SYSTEM distributed_example
  (* Version 1.0, 2025-11-18, obotnar *)
  APPLICATION distributed_exampleApp
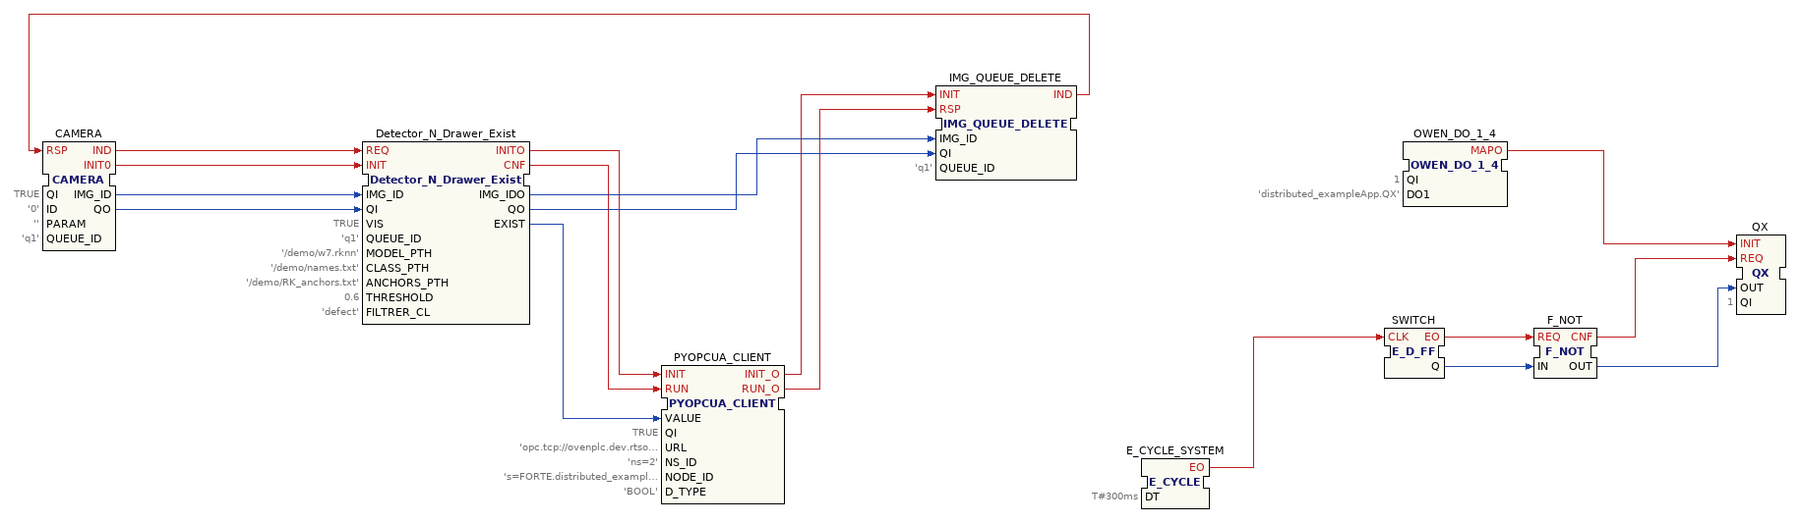
    FBS
      CAMERA : CAMERA(QI := TRUE, ID := '0', PARAM := '', QUEUE_ID := 'q1');
      IMG_QUEUE_DELETE : IMG_QUEUE_DELETE(QUEUE_ID := 'q1');
      Detector_N_Drawer_Exist : Detector_N_Drawer_Exist(VIS := TRUE, QUEUE_ID := 'q1', MODEL_PTH := '/demo/w7.rknn', CLASS_PTH := '/demo/names.txt', ANCHORS_PTH := '/demo/RK_anchors.txt', THRESHOLD := 0.6, FILTRER_CL := 'defect');
      PYOPCUA_CLIENT : PYOPCUA_CLIENT(QI := TRUE, URL := 'opc.tcp://ovenplc.dev.rtsoft.ru:4843', NS_ID := 'ns=2', NODE_ID := 's=FORTE.distributed_exampleApp.SWITCH.D', D_TYPE := 'BOOL');
      E_CYCLE_SYSTEM : E_CYCLE(DT := T#300ms);
      QX : QX(QI := 1 {SET_ATTRIBUTE(OpcMapping, true)}, PARAMS :=  {SET_ATTRIBUTE(OpcMapping, true)}, OUT :=  {SET_ATTRIBUTE(OpcMapping, true)}, QO :=  {SET_ATTRIBUTE(OpcMapping, true)}, STATUS :=  {SET_ATTRIBUTE(OpcMapping, true)});
      OWEN_DO_1_4 : OWEN_DO_1_4(QI := 1 {SET_ATTRIBUTE(OpcMapping, true)}, DO1 := 'distributed_exampleApp.QX' {SET_ATTRIBUTE(OpcMapping, true)}, DO2 :=  {SET_ATTRIBUTE(OpcMapping, true)}, DO3 :=  {SET_ATTRIBUTE(OpcMapping, true)}, DO4 :=  {SET_ATTRIBUTE(OpcMapping, true)}, QO :=  {SET_ATTRIBUTE(OpcMapping, true)}, STATUS :=  {SET_ATTRIBUTE(OpcMapping, true)});
      SWITCH : E_D_FF(D :=  {SET_ATTRIBUTE(OpcMapping, true)}, Q :=  {SET_ATTRIBUTE(OpcMapping, true)});
      F_NOT : F_NOT;
    END_FBS
    EVENT_CONNECTIONS
      CAMERA.IND TO Detector_N_Drawer_Exist.REQ;
      CAMERA.INIT0 TO Detector_N_Drawer_Exist.INIT;
      Detector_N_Drawer_Exist.INITO TO PYOPCUA_CLIENT.INIT;
      PYOPCUA_CLIENT.INIT_O TO IMG_QUEUE_DELETE.INIT;
      Detector_N_Drawer_Exist.CNF TO PYOPCUA_CLIENT.RUN;
      E_CYCLE_SYSTEM.EO TO SWITCH.CLK;
      OWEN_DO_1_4.MAPO TO QX.INIT;
      PYOPCUA_CLIENT.RUN_O TO IMG_QUEUE_DELETE.RSP;
      SWITCH.EO TO F_NOT.REQ;
      F_NOT.CNF TO QX.REQ;
      IMG_QUEUE_DELETE.IND TO CAMERA.RSP;
    END_CONNECTIONS
    DATA_CONNECTIONS
      CAMERA.IMG_ID TO Detector_N_Drawer_Exist.IMG_ID;
      Detector_N_Drawer_Exist.IMG_IDO TO IMG_QUEUE_DELETE.IMG_ID;
      CAMERA.QO TO Detector_N_Drawer_Exist.QI;
      Detector_N_Drawer_Exist.QO TO IMG_QUEUE_DELETE.QI;
      Detector_N_Drawer_Exist.EXIST TO PYOPCUA_CLIENT.VALUE;
      F_NOT.OUT TO QX.OUT;
      SWITCH.Q TO F_NOT.IN;
    END_CONNECTIONS
  END_APPLICATION
  DEVICE FORTE_PC : FORTE_PC(MGR_ID := "10.5.20.137:62499" (* Device manager socket ID *))
    {SET_ATTRIBUTE(Profile, HOLOBLOC)}
    RESOURCE EMB_RES : EMB_RES
    END_RESOURCE
  END_DEVICE
  DEVICE FORTE_PC_1 : FORTE_PC(MGR_ID := "10.5.20.68:61499" (* Device manager socket ID *))
    {SET_ATTRIBUTE(Profile, HOLOBLOC)}
    RESOURCE FLOGIC_EMB_RES : FLOGIC_EMB_RES(ENABLE_RETAIN :=  (* Enable retain in resource *), OPC_BASE_PATH :=  (* Path to base OPCUA node *))
      EVENT_CONNECTIONS
        START.COLD TO distributed_exampleApp.OWEN_DO_1_4.MAP;
        START.WARM TO distributed_exampleApp.OWEN_DO_1_4.MAP;
        START.COLD TO distributed_exampleApp.E_CYCLE_SYSTEM.START;
        START.WARM TO distributed_exampleApp.E_CYCLE_SYSTEM.START;
        START.STOP TO distributed_exampleApp.E_CYCLE_SYSTEM.STOP;
        distributed_exampleApp.E_CYCLE_SYSTEM.EO TO OPCUAS.REQ;
      END_CONNECTIONS
    END_RESOURCE
  END_DEVICE
  MAPPINGS
    distributed_exampleApp.E_CYCLE_SYSTEM ON FORTE_PC_1.FLOGIC_EMB_RES;
    distributed_exampleApp.QX ON FORTE_PC_1.FLOGIC_EMB_RES;
    distributed_exampleApp.SWITCH ON FORTE_PC_1.FLOGIC_EMB_RES;
    distributed_exampleApp.OWEN_DO_1_4 ON FORTE_PC_1.FLOGIC_EMB_RES;
    distributed_exampleApp.CAMERA ON FORTE_PC.EMB_RES;
    distributed_exampleApp.Detector_N_Drawer_Exist ON FORTE_PC.EMB_RES;
    distributed_exampleApp.PYOPCUA_CLIENT ON FORTE_PC.EMB_RES;
    distributed_exampleApp.IMG_QUEUE_DELETE ON FORTE_PC.EMB_RES;
    distributed_exampleApp.F_NOT ON FORTE_PC_1.FLOGIC_EMB_RES;
  END_MAPPINGS
END_SYSTEM
